{attribute 'linkalways'} 
{attribute 'no_explicit_call' := 'This FB is a CLASS and must be accessed using methods or properties'}
{attribute 'enable_dynamic_creation'}
FUNCTION_BLOCK VisionDatatypePack IMPLEMENTS I_DatatypePack
VAR
	// alias
	
	// enums
	_eTcVn2dCodeSearchStrategy : _ETcVn2dCodeSearchStrategy(ETcVn2dCodeSearchStrategy.TCVN_CSS_DEFAULT);
	
	// structures
	
END_VAR

METHOD RegisterWith
VAR_INPUT
	Datatypes : I_Datatypes;
END_VAR
Datatypes.RegisterDatatype(_eTcVn2dCodeSearchStrategy);
END_METHOD

END_FUNCTION_BLOCK

(* stored: Version 1.1.0.1
   POU VisionDatatypePack: Id {faa9ad1a-2b24-4d20-95e0-67a7c7e3da9c}, SpecialFunc None
   Method RegisterWith: Id {e0f84940-a921-4fc9-8944-9e8dd00778cd} *)
